FUNCTION_BLOCK FB_AxisControl
VAR_INPUT
	xEnable: BOOL;
	xZero: BOOL;
	xMoveR: BOOL;
	xMoveA: BOOL;
	xMoveV: BOOL;
	xPositiveDirection: BOOL;
	fDistance: LREAL;
	fPosition: LREAL;
	fVelocity: LREAL;
	xStop: BOOL;
	xHome: BOOL;
	fHomeOffset: LREAL;
	xHomeFlag: BOOL;
END_VAR
VAR_OUTPUT
	fActualPosition: LREAL;
	fActualVelocity: LREAL;
	fActModuloPos: LREAL;
	xEnabled: BOOL;
	xMoveComplete: BOOL;
	xInPosition: BOOL;
	xAtSpeed: BOOL;
	xStopped: BOOL;
	xHomed: BOOL;
	stStatus : ST_AxisStatus;
	CommandAborted : BOOL;
	bStandStill : BOOL;
END_VAR
VAR
	mcPower: MC_Power;
	mcReset: MC_Reset;
	mcMoveRelative: MC_MoveRelative;
	mcSetPosition: MC_SetPosition;
	mcMoveAbsolute: MC_MoveAbsolute;
	mcReadStatus: MC_ReadStatus;
	mcMoveVelocity: MC_MoveVelocity;
	mcStop: MC_Stop;
	mcHome: MC_Home;
END_VAR
VAR_IN_OUT
	Axis: AXIS_REF;
END_VAR

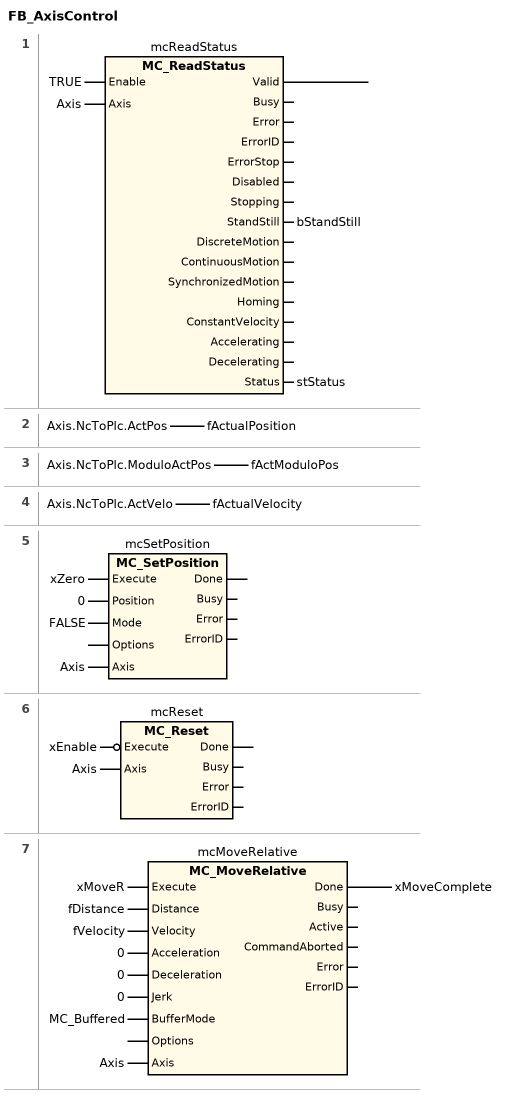
// NETWORK 1
mcReadStatus(Enable := TRUE, Axis := Axis, StandStill => bStandStill, Status => stStatus); // MC_ReadStatus

// NETWORK 2
fActualPosition := Axis.NcToPlc.ActPos;

// NETWORK 3
fActModuloPos := Axis.NcToPlc.ModuloActPos;

// NETWORK 4
fActualVelocity := Axis.NcToPlc.ActVelo;

// NETWORK 5
mcSetPosition(Execute := xZero, Position := 0, Mode := FALSE, Axis := Axis); // MC_SetPosition

// NETWORK 6
mcReset(Execute := NOT xEnable, Axis := Axis); // MC_Reset

// NETWORK 7
mcMoveRelative(
    Execute := xMoveR,
    Distance := fDistance,
    Velocity := fVelocity,
    Acceleration := 0,
    Deceleration := 0,
    Jerk := 0,
    BufferMode := MC_Buffered,
    Axis := Axis); // MC_MoveRelative
xMoveComplete := mcMoveRelative.Done;

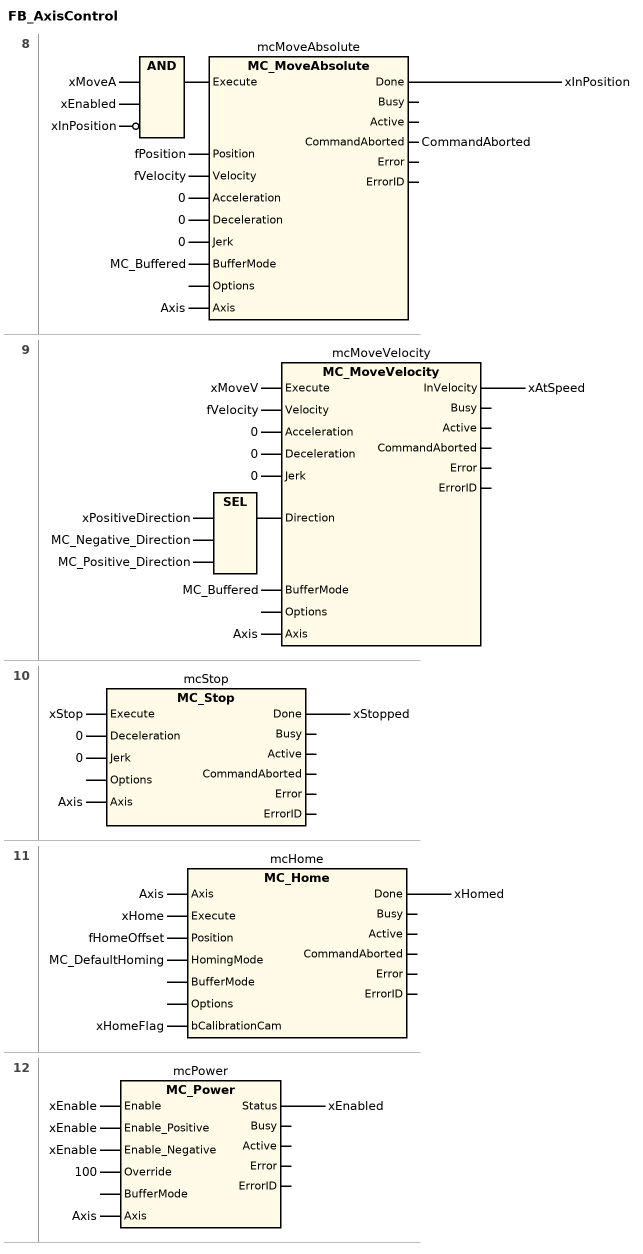
// NETWORK 8
mcMoveAbsolute(
    Execute := xMoveA AND xEnabled AND NOT xInPosition,
    Position := fPosition,
    Velocity := fVelocity,
    Acceleration := 0,
    Deceleration := 0,
    Jerk := 0,
    BufferMode := MC_Buffered,
    Axis := Axis,
    CommandAborted => CommandAborted); // MC_MoveAbsolute
xInPosition := mcMoveAbsolute.Done;

// NETWORK 9
mcMoveVelocity(
    Execute := xMoveV,
    Velocity := fVelocity,
    Acceleration := 0,
    Deceleration := 0,
    Jerk := 0,
    Direction := SEL(xPositiveDirection, MC_Negative_Direction, MC_Positive_Direction),
    BufferMode := MC_Buffered,
    Axis := Axis); // MC_MoveVelocity
xAtSpeed := mcMoveVelocity.InVelocity;

// NETWORK 10
mcStop(Execute := xStop, Deceleration := 0, Jerk := 0, Axis := Axis); // MC_Stop
xStopped := mcStop.Done;

// NETWORK 11
mcHome(
    Axis := Axis,
    Execute := xHome,
    Position := fHomeOffset,
    HomingMode := MC_DefaultHoming,
    bCalibrationCam := xHomeFlag); // MC_Home
xHomed := mcHome.Done;

// NETWORK 12
mcPower(
    Enable := xEnable,
    Enable_Positive := xEnable,
    Enable_Negative := xEnable,
    Override := 100,
    Axis := Axis); // MC_Power
xEnabled := mcPower.Status;

END_FUNCTION_BLOCK

(* stored: Version 1.1.0.1, ProductVersion 3.1.4024.4
   POU FB_AxisControl: Id {f227cd92-c705-4204-9270-5ec21594e959}, SpecialFunc None *)
